{attribute 'qualified_only'}
VAR_GLOBAL CONSTANT
	MaxStepCount : INT := 5;	
	MaxStepActionsCount : INT := 5;
	MaxStepTransitionsCount : INT := 2;
	MaxActionArgumentsCount : INT := 5;
	MaxConditionArgumentsCount : INT := 5;
END_VAR

(* stored: Version 1.1.0.1
   GVL UnifiedProgramConstants: Id {948c2321-8227-45fd-9533-ace11dca37a6} *)
